Staubli VAL3: addDirectory.pgx

public program addDirectory(bool& x_bRe, string x_sPath, string x_sDirName)
  local bool l_bool1
  local num l_i
begin
  //建立一个文件夹
  x_bRe=libList("Disk://",sContent)
  if !x_bRe
    return
  endIf

  if sContent[0]!=""
    x_bRe=$copy("Disk://"+sContent[0],x_sPath+"/"+x_sDirName)
    if !x_bRe
      return
    endIf
    x_bRe=libList(x_sPath+"/"+x_sDirName,sContent)
    if !x_bRe
      return
    endIf
    for l_i=0 to size(sContent)-1
      if sContent[l_i]!=""
        x_bRe=$delete(x_sPath+"/"+x_sDirName+"/"+sContent[l_i])
        if !x_bRe
          return
        endIf
      endIf
    endFor
  endIf
end
